KUKA KRL program: chk_w3_grp3_opn.src

&ACCESS RVO1
&COMMENT Check GRP Z3 ACTROS OPEN
DEF chk_w3_grp3_opn( )

; Check gripper actros OPEN Z3
;//---- Start User-------

$TIMER[10] = 0
$TIMER_STOP[10] = FALSE

WAIT FOR (NOT $IN[12])
WAIT FOR ($IN[11])

$TIMER_STOP[10] = TRUE
$TIMER[10] = 0

;//---- End User---------

END
